PROGRAM Version
VAR
END_VAR

(*
1.0.1.1:	Boido	010120

Changed naming convention for main modules.
The first 2 letters give a hint on the inheritance relationship of the FB.

1.0.2.2:	Boido	010120

Naming convention adjustments.

1.1.0.3:	Boido	010120

Every IO variable is of type BoolIn or BoolOut.
In the future when different types will be needed,
also RealIn,RealOut,IntIn,IntOut etc.. will be added.

1.1.1.4:	Boido	010120

New StepWorkerLib v:1033, naming conventions fixes and IO adjustments

1.1.2.5:	Boido	020120

Version.txt replaced with Version PRG

*)

END_PROGRAM

(* stored: Version 1.1.0.1, ProductVersion 3.1.4024.0
   POU Version: Id {c0e64eec-c0cd-4b22-8e7a-7dec7d9bd2c8}, SpecialFunc None *)
